TYPE U_BytesToWord :
UNION
	arByteIn:ARRAY [0..1] OF BYTE;
	uintOut: UINT;
END_UNION
END_TYPE

(* stored: Version 1.1.0.1, ProductVersion 3.1.4024.9
   DUT U_BytesToWord: Id {5948d70f-820c-4cff-864a-288dfddfd688} *)
